FUNCTION_BLOCK Test_Raises_OnDaysChanged EXTENDS TUnitTestBase
IMPLEMENTS 
    IEventHandler_OnDayChanged
VAR
    NowFromEvent : TIMESTRUCT;
    
    OnDaysChanged_Raised    : BOOL;
END_VAR

METHOD  Execute
VAR_INST
    ClockEventSource : TClockEventSource;
    Now              : TIMESTRUCT := (wDay := 23, wMonth := 12, wYear := 1945, wHour := 22, wMinute := 20, wSecond := 18);
    OneDayLater      : TIMESTRUCT := (wDay := 24, wMonth := 12, wYear := 1945, wHour := 22, wMinute := 20, wSecond := 18);
END_VAR
OnDaysChanged_Raised := FALSE;

ClockEventSource.Event_DayChanged.ClearEventHandlers().AddEventHandler(THIS^);

ClockEventSource.Init(Now := Now);
ClockEventSource(Now := OneDayLater);

Assertion.AssertEquals_BOOL(
    Expected := TRUE,
    Actual   := OnDaysChanged_Raised,
    ObjectName := _TestName,
    VariableName  := 'OnDaysChanged_Raised');

Assertion.AssertEquals_STRUCT(
    Expected := OneDayLater,
    Actual   := NowFromEvent,
    ObjectName := _TestName,
    VariableName  := 'NowFromEvent');

Test_Finished();
END_METHOD

METHOD OnDayChanged
VAR_INPUT
	Now	: Tc2_Utilities.TIMESTRUCT;
END_VAR
NowFromEvent := Now;
OnDaysChanged_Raised := TRUE;
END_METHOD

END_FUNCTION_BLOCK

(* stored: Version 1.1.0.1, ProductVersion 3.1.4024.3
   POU Test_Raises_OnDaysChanged: Id {dadfe947-d3e3-0cc8-2098-8ccd5150a4f2}, SpecialFunc None
   Method Execute: Id {9bd40728-3acd-0754-09ad-f6d44c7fb0a9}
   Method OnDayChanged: Id {cdd1c03d-8054-017d-2eec-f1bfc76bc907} *)
